// TIA Portal V17 export
// export: Created 2025-03-05T08:02:27.524743Z, ExportSetting WithDefaults, DisplayName Totally Integrated Automation Portal, DisplayVersion V17 Update 8, DisplayName TIA Portal Openness, DisplayVersion V17 Update 8, DisplayName TIA Portal Version Control Interface, DisplayVersion V17, DisplayName SINAMICS Startdrive Advanced, DisplayVersion V17 SP2, DisplayName SINAMICS Startdrive G110M, G120, G120C, G120D, G120P, G115D, DisplayVersion V17 SP2, DisplayName SINAMICS Startdrive G130, G150, S120, S150, SINAMICS MV, S210, DisplayVersion V17 SP2, DisplayName STEP 7 Professional, DisplayVersion V17 Update 8, DisplayName SINUMERIK ONE STEP 7 Toolbox, DisplayVersion V17 Update 12, DisplayName SINUMERIK 840D sl STEP 7 Toolbox, DisplayVersion V17 Update 12, DisplayName STEP 7 Safety, DisplayVersion V17 Update 6, DisplayName WinCC Advanced, DisplayVersion V17 Update 8
TYPE "LASER TRUMPF"
// stored: IsFailsafeCompliant false
   STRUCT
      OUTPUTS : Struct
         CONTROL : Struct
            LASER_REQUEST : Bool := FALSE;   // REQUESTING THE LASER
            PILOT_LASER_ON : Bool := FALSE;   // SWITCHING ON THE PILOT LASER
            UNSYNC_PSTART : Bool := FALSE;   // UNSYNCHRONIZED ACTIVATION
            SIMULATION : Bool := FALSE;   // SIMULATION MODE
            LOCK_PROG_PARAM : Bool := FALSE;   // ONLY FOR TRUMICRO: LOCK OPERATING POINT PARAMETERS. RESERVED FOR ALL OTHER LASER DEVICES.
            INQUIRY_2 : Bool := FALSE;   // QUERY INPUT 2
            INQUIRY_1 : Bool := FALSE;   // QUERY INPUT 1
            FAULT_EXTERNAL : Bool := FALSE;   // EXTERNAL FAULT
            RESET : Bool := FALSE;   // RESET
            PROGRAM_STOP : Bool := FALSE;   // CANCEL / STOP LASER PROGRAM
            PROG_START_DYN : Bool := FALSE;   // DYNAMIC PROGRAM START
            PROG_START_SATICAL : Bool := FALSE;   // STATIC PROGRAM START
            LASER_STANDBY : Bool := FALSE;   // ACTIVATING THE LASER STANDBY MODE
            LASER_ON : Bool := FALSE;   // SWITCHING ON THE LASER
            LOCK_OPERAT_PANEL : Bool := FALSE;   // LOCKING THE OPERATING PANE
            EXT_CONTROL : Bool := FALSE;   // EXTERNAL CONTROL
         END_STRUCT;
         PROGRAMNO : Byte := B#16#0;   // NUMBER OF THE SELECTED LASER PROGRAM
         LIGHTPATH : Byte := B#16#0;   // NUMBER OF THE SELECTED LIGHT PATH
         LASER_NO : Byte := B#16#0;   // NUMBER OF THE SELECTED LASER DEVICE
         AD_NO : Byte := B#16#0;   // NUMBER OF THE APPLICATION DATA SET
         POWER_VALUE : Word := W#16#0;   // POWER VALUE (IW3)
         PROCESSING : Word := W#16#0;   // PROCESSING (IW4)
         POWER_PORTION_CORE : Word;   // POWER PORTION CORE (IW5)
      END_STRUCT;
      INPUTS : Struct
         STATUS : Struct
            LASER_WARNING_LAP_ON : Bool := FALSE;   // THE LASER WARNING LIGHT IS ON
            PILOT_LASER_IS_ON : Bool := FALSE;   // PILOT LASER IS SWITCHED ON
            POWER_LIMIT : Bool := FALSE;   // THE POWER LIMIT OF THE LASER HAS BEEN REACHED
            LASER_ASSIGNED : Bool := FALSE;   // THE LASER DEVICE IS ASSIGNED TO AN EXTERNAL CONTROL UNIT
            FAULT_LASER : Bool := FALSE;   // A FAULT MESSAGE OF THE LASER DEVICE IS ACTIVE
            MONITORING : Bool := FALSE;   // A MONITORING MESSAGE OF THE LASER DEVICE IS ACTIVE
            SIK_OPEN : Bool := FALSE;   // THE SAFETY CIRCUIT (SIK) IS OPEN
            SET_3 : Bool := FALSE;   // SET OUTPUTS 3
            SET_2 : Bool := FALSE;   // SET OUTPUTS 2
            SET_1 : Bool := FALSE;   // SET OUTPUTS 1
            PROG_CANCELED : Bool := FALSE;   // LASER PROGRAM HAS BEEN CANCELLED
            PROG_COMPLETED : Bool := FALSE;   // LASER PROGRAM IS COMPLETED
            PROG_ACTIVE : Bool := FALSE;   // LASER PROGRAM IS ACTIVE
            LASER_READY : Bool := FALSE;   // THE LASER OF THE LASER DEVICE IS READY
            LASER_IS_ON : Bool := FALSE;   // THE LASER OF THE LASER DEVICE IS SWITCHED ON
            EXT_ACTIV_ACTIVE : Bool := FALSE;   // EXTERNAL ACTIVATION IS ACTIVE
         END_STRUCT;
         PROGRAMNO_ACK : Byte := B#16#0;   // ACKNOWLEDGEMENT OF THE NUMBER OF THE LASER PROGRAMSELECTED
         LIGHTPATH_ACK : Byte := B#16#0;   // ACKNOWLEDGEMENT OF THE NUMBER OF THE CURRENTLY SET LIGHTPATH
         SHUTTER_SWITCH_1 : Bool;   // POSITION OF THE SHUTTER SWITCHES
         SHUTTER_SWITCH_2 : Bool;   // POSITION OF THE SHUTTER SWITCHES
         SHUTTER_SWITCH_3 : Bool;   // POSITION OF THE SHUTTER SWITCHES
         SHUTTER_SWITCH_4 : Bool;   // POSITION OF THE SHUTTER SWITCHES
         SHUTTER_SWITCH_5 : Bool;   // POSITION OF THE SHUTTER SWITCHES
         SHUTTER_SWITCH_6 : Bool;   // POSITION OF THE SHUTTER SWITCHES
         SHUTTER_SWITCH_7 : Bool;   // POSITION OF THE SHUTTER SWITCHES
         SHUTTER_SWITCH_8 : Bool;   // POSITION OF THE SHUTTER SWITCHES
         FAULT_SLOT : Bool := FALSE;   // A LOCAL FAULT HAS OCCURRED FOR THIS SLOT
         MONITORING_SLOT : Bool := FALSE;   // A LOCAL MONITORING HAS OCCURRED FOR THIS SLOT
         RESERVED_1 : Bool := FALSE;   // RESERVE
         OPTICS_AVAILABLE : Bool := FALSE;   // FOCUSING OPTICS OR LIGHT PATH COMPONENT IS ENABLED.
         OPTICS_READY : Word;   // THE FOCUSING OPTICS OR LIGHT PATH COMPONENT IS READY FOR OPERATION.
         VALUES_IN_RANGE : Bool := FALSE;   // APPLICATION VALUES CROSSJET PRESSURE, EXHAUSTION AND SHIELDING GAS ARE IN THE ADMISSIBLE RANGE
         PROT_GLASS_CONTAM : Bool := FALSE;   // LIMIT VALUE MAX1 OF THE PROTECTIVE GLASS CONTAMINATION HASBEEN REACHED
         PROT_GLASS_LIFE_RCHD : Bool := FALSE;   // LIMIT VALUE MAX2 OF THE PROTECTIVE GLASS CONTAMINATION HASBEEN REACHED
         MEAS_VAL_OUT_ACT : Bool := FALSE;   // OUTPUT WORD 4 OUTPUTS MEASURED VALUE ID
         MAINTENACE : Bool := FALSE;   // MAINTENANCE OF THE LASER DEVICE IS REQUIRED
         RESERVED_2 : Bool;   // RESERVE
         CALIBRATION : Bool := FALSE;   // THE LASER IS BEING CALIBRATED OR LASER SELFTEST IS ACTIVE
         ALIVE_TICK : Bool := FALSE;   // LASER CONTROL IS ACTIVE
         EXT_COOL_ON : Bool := FALSE;   // EXTERNAL COOLING CIRCUIT IS SWITCHED ON OR THE LASER DEVICE REQUIRES COOLING WATER
         RESERVED_3 : Bool;   // RESERVE
         RESERVED_4 : Bool;   // RESERVE
         LASER_NO_1 : Bool;   // NUMBER OF THE LASER DEVICE BIT 1
         LASER_NO_2 : Bool;   // NUMBER OF THE LASER DEVICE BIT 2
         LASER_NO_3 : Bool;   // NUMBER OF THE LASER DEVICE BIT 3
         LASER_NO_4 : Bool;   // NUMBER OF THE LASER DEVICE BIT 4
         LASER_NO_5 : Bool;   // NUMBER OF THE LASER DEVICE BIT 5
         LASER_NO_6 : Bool;   // NUMBER OF THE LASER DEVICE BIT 6
         LASER_NO_7 : Bool;   // NUMBER OF THE LASER DEVICE BIT 7
         LASER_NO_8 : Bool;   // NUMBER OF THE LASER DEVICE BIT 8
         MESSAGE_NUM : Byte;   // MESSAGE CODE NUM
         MESSAGE_ID : Byte;   // MESSAGE CODE ID
         MESSAGE_CODE : Word;   // MESSAGE CODE OF THE REPORTING COMPONENT
         LASER_POWER : Word;   // CW LASER: LASER POWER
         ENERGY : Word;   // PULSE ENERGY
         RESERVED_WORD_8 : Word;   // RESERVE WORD
      END_STRUCT;
   END_STRUCT;
END_TYPE
